{attribute 'qualified_only'}
VAR_GLOBAL

	//HSS
	TempDIDSupPrim			:	REAL;
	TempDIDRetPrim			:	REAL;
	TempDIDSup				:	REAL;
	TempDIDRet				:	REAL;
	
	
END_VAR

(* stored: Version 1.1.0.1, ProductVersion 3.1.4024.3
   GVL TempSensors: Id {85ca2fa2-2375-48f1-a6ce-727919266df1} *)
